{attribute 'qualified_only'}
{attribute 'strict'}
{attribute 'to_string'}
TYPE systemStatus_t :
(
	STOPPED := 0,
	STARTING := 1,
	RUNNING := 2,
	ERROR := 3,
	STOPPING := 4
);
END_TYPE

(* stored: Version 1.1.0.1
   EnumerationTextList systemStatus_t: Id {e0f12b2e-f9e3-4ce9-b84b-9dc2c70e8af5} *)
